{attribute 'GeneratedUsingTerminal: IndraDrive MPB20-0003-0000'}
{attribute addProperty BoxType "IndraDrive MPB20-0003-0000"}
{attribute addProperty Id "Drive_status_wordAT %I*UINT2Position_feedback_value_1AT %I*DINT4"}
{attribute addProperty CRC "650925181"}
{attribute addProperty Size "6"}
TYPE AT_x_26CC547D EXTENDS TcoIo.InputBase_8311D824 : 
STRUCT
    {attribute addProperty Name "Drive_status_word"}
    Drive_status_word AT %I* : UINT;
    {attribute addProperty Name "Position_feedback_value_1"}
    Position_feedback_value_1 AT %I* : DINT;
END_STRUCT
END_TYPE

(* stored: Version 1.2.0.0, ProductVersion 3.1.4024.11
   DUT AT_x_26CC547D: Id {15defaa8-68b7-049d-0908-bec4be166d62} *)
